(* IEC 61131-3 sources: POMIRTS_lab3/AS/Library_2/LoopCont/V2.12.0, 3 files *)

(* ---- LoopCont.typ ---- *)
(********************************************************************
 * COPYRIGHT (C) BERNECKER + RAINER, AUSTRIA, A-5142 EGGELSBERG
 ********************************************************************
 * Library: LoopCont
 * File: LoopCont.typ
 * Created: 11.11.2003
 ********************************************************************
 * Global data types of library LoopCont
 ********************************************************************)
TYPE
	lcCurveByPoints_TabEntry_type : STRUCT
		x	: INT ;
		y	: INT ;
	END_STRUCT;
	lcpid_addPar_typ : STRUCT
		y_autotune_on	: INT ;
		y_autotune_off	: INT ;
		t_autotune_max	: UDINT ;
		diff_dx_max	: INT ;
		diff_dt_max	: UDINT ;
		osc_nrPeriods	: UINT ;
		osc_minAmplitude	: INT ;
		optSwitches	: UINT ;
		dY_max	: REAL ;
		Tf_Tv	: REAL ;
		Kw	: REAL ;
		Kfbk	: REAL ;
		fbk_mode	: USINT ;
		d_mode	: USINT ;
		calc_mode	: USINT ;
	END_STRUCT;
	lcpid_internal_typ : STRUCT
		size	: UINT ;
		valid	: BOOL ;
		autotune_addpar	: lcpid_addPar_typ ;
		Y_max	: INT ;
		Y_min	: INT ;
		dY_max1	: DINT ;
		Kp1	: DINT ;
		Kp_Tn_1	: DINT ;
		Tv_Tf_1	: DINT ;
		Tf_reciproc_1	: DINT ;
		Kw1	: DINT ;
		Kfbk_Kp_1	: DINT ;
		fbk_mode	: USINT ;
		d_mode	: USINT ;
		calc_mode	: USINT ;
		prescalerPow2	: UINT ;
		force_outmode	: USINT ;
		Y_force	: INT ;
		W	: INT ;
		X	: INT ;
		pid_init	: USINT ;
		dt	: UDINT ;
		Yp1	: DINT ;
		Yp2	: DINT ;
		dYi1	: DINT ;
		dYi2	: DINT ;
		Yi1	: DINT ;
		Yi2	: DINT ;
		dt_Tf_1	: DINT ;
		a11	: DINT ;
		a12	: DINT ;
		a21	: DINT ;
		a22	: DINT ;
		Yd1	: DINT ;
		Yd2	: DINT ;
		Ytotal1	: DINT ;
		Ytotal2	: DINT ;
		Ylim1	: DINT ;
		Ylim2	: DINT ;
		Y1	: DINT ;
		Y2	: DINT ;
		e_fbk	: DINT ;
	END_STRUCT;
	lcpid_osc_val_typ : STRUCT
		X	: INT ;
		t	: UDINT ;
	END_STRUCT;
	lcpid_osc_per_typ : STRUCT
		max	: lcpid_osc_val_typ ;
		min	: lcpid_osc_val_typ ;
	END_STRUCT;
	lcpid_osc_typ : STRUCT
		i_maxPeriod	: UINT ;
		i_period	: UINT ;
		X_amplitude	: DINT ;
		amplitudeRatio	: REAL ;
		tPeriod	: UDINT ;
		period	: ARRAY[0..4] OF lcpid_osc_per_typ ;
	END_STRUCT;
	lcpid_procPar_typ : STRUCT
		size	: UINT ;
		stepResp_valid	: BOOL ;
		stepResp_v	: REAL ;
		stepResp_t_u	: UDINT ;
		osc_valid	: BOOL ;
		osc_amplitudeRatio	: REAL ;
		osc_tPeriod	: UDINT ;
		force_params	: BOOL ;
		Kp	: REAL ;
		Tn	: REAL ;
		Tv	: REAL ;
	END_STRUCT;
	lcpid_old_typ : STRUCT
		processPar	: lcpid_procPar_typ ;
		P_manualAdjust	: INT ;
		I_manualAdjust	: INT ;
		D_manualAdjust	: INT ;
		Y_min	: INT ;
		Y_max	: INT ;
		dY_max	: REAL ;
		Kw	: REAL ;
		Kfbk	: REAL ;
		enable	: BOOL ;
		request	: USINT ;
		time	: UDINT ;
	END_STRUCT;
	lcpid_stepResp_typ : STRUCT
		W_old	: INT ;
		dW	: INT ;
		x_prev	: INT ;
		x_inflectionPt	: INT ;
		t_inflectionPt	: UDINT ;
		v	: REAL ;
		v_max	: REAL ;
		t_u	: UDINT ;
		x_pre	: INT ;
		x_max	: INT ;
	END_STRUCT;
	lcpid_diff_typ : STRUCT
		init	: BOOL ;
		x_old	: INT ;
		dx	: INT ;
		dt	: UDINT ;
		dx_dt	: REAL ;
	END_STRUCT;
END_TYPE

(* ---- LoopCont.fun ---- *)
(********************************************************************
 * COPYRIGHT (C) BERNECKER + RAINER, AUSTRIA, A-5142 EGGELSBERG
 ********************************************************************
 * Library: LoopCont
 * File: LoopCont.fun
 * Created: 11.11.2003
 ********************************************************************
 * Functions and function blocks of library LoopCont
 ********************************************************************)
FUNCTION_BLOCK LCCurveByPoints
	VAR_INPUT
		x	:INT;
		NoOfPoints	:UINT;
		ptr_table	:REFERENCE TO lcCurveByPoints_TabEntry_type;
	END_VAR
	VAR_OUTPUT
		status	:UINT;
		y	:INT;
	END_VAR
	VAR
		i_tab	:INT;
		iterations	:UINT;
		scal1	:LCScINT;
	END_VAR
END_FUNCTION_BLOCK
FUNCTION_BLOCK LCPWM_DMod
	VAR_INPUT
		enable	:BOOL;
		x	:INT;
		max_value	:INT;
		min_value	:INT;
		tminpuls	:UINT;
		tperiod	:UINT;
		basetime	:UDINT;
	END_VAR
	VAR_OUTPUT
		status	:UINT;
		y	:BOOL;
	END_VAR
	VAR
		area	:DINT;
		period	:UINT;
		time_old	:UDINT;
		last	:UINT;
		x_old	:INT;
		enable_old	:BOOL;
	END_VAR
END_FUNCTION_BLOCK
FUNCTION_BLOCK LCPIDpara
	VAR_INPUT
		enable	:BOOL;
		enter	:BOOL;
		Y_max	:INT;
		Y_min	:INT;
		dY_max	:REAL;
		Kp	:REAL;
		Tn	:REAL;
		Tv	:REAL;
		Tf	:REAL;
		Kw	:REAL;
		Kfbk	:REAL;
		fbk_mode	:USINT;
		d_mode	:USINT;
		calc_mode	:USINT;
	END_VAR
	VAR_OUTPUT
		status	:UINT;
		ident	:UDINT;
	END_VAR
	VAR
		internal_data	:lcpid_internal_typ;
	END_VAR
END_FUNCTION_BLOCK
FUNCTION_BLOCK LCRampLim
	VAR_INPUT
		enable	:BOOL;
		x	:INT;
		tup	:UINT;
		tdown	:UINT;
		max_value	:INT;
		min_value	:INT;
		yset	:INT;
		set	:BOOL;
		basetime	:UDINT;
	END_VAR
	VAR_OUTPUT
		status	:UINT;
		y	:INT;
		xreached	:BOOL;
		max_limit	:BOOL;
		min_limit	:BOOL;
	END_VAR
	VAR
		time_old	:UDINT;
		rest	:UINT;
		enable_old	:BOOL;
	END_VAR
END_FUNCTION_BLOCK
FUNCTION_BLOCK LCPID
	VAR_INPUT
		enable	:BOOL;
		ident	:UDINT;
		W	:INT;
		X	:INT;
		A	:INT;
		Y_man	:INT;
		Y_fbk	:INT;
		hold_I	:BOOL;
		out_mode	:USINT;
		basetime	:UDINT;
	END_VAR
	VAR_OUTPUT
		status	:UINT;
		e	:DINT;
		Y	:INT;
		Yp	:DINT;
		Yi	:DINT;
		Yd	:DINT;
	END_VAR
	VAR
		time_old	:UDINT;
		Tv_Tf_old	:DINT;
		enable_old	:BOOL;
		e_old	:DINT;
	END_VAR
END_FUNCTION_BLOCK
FUNCTION_BLOCK LCTimeBasedOnOff
	VAR_INPUT
		enable	:BOOL;
		x	:INT;
		max_value	:INT;
		min_value	:INT;
		timpulse	:UINT;
		tchange_up	:UINT;
		tchange_dwn	:UINT;
		ref	:BOOL;
		basetime	:UDINT;
	END_VAR
	VAR_OUTPUT
		status	:UINT;
		up	:BOOL;
		down	:BOOL;
		hysteresis_up	:UINT;
		hysteresis_dwn	:UINT;
		refOK	:BOOL;
	END_VAR
	VAR
		time_old	:UDINT;
		ref_old	:BOOL;
		t_cnt	:DINT;
		y_fix31_1	:DINT;
		y_fix31_2	:DINT;
	END_VAR
END_FUNCTION_BLOCK
FUNCTION_BLOCK LCDifferentiate
	VAR_INPUT
		enable	:BOOL;
		x	:INT;
		tv	:UINT;
		tf	:UINT;
		basetime	:UDINT;
	END_VAR
	VAR_OUTPUT
		status	:UINT;
		y	:INT;
	END_VAR
	VAR
		time_old	:UDINT;
		enable_old	:BOOL;
		a2n	:DINT;
		a1	:DINT;
	END_VAR
END_FUNCTION_BLOCK
FUNCTION_BLOCK LCPIDAutoTune
	VAR_INPUT
		enable	:BOOL;
		Y_max	:INT;
		Y_min	:INT;
		P_manualAdjust	:INT;
		I_manualAdjust	:INT;
		D_manualAdjust	:INT;
		request	:USINT;
		basetime	:UDINT;
	END_VAR
	VAR_OUTPUT
		status	:UINT;
		ident	:UDINT;
		addInfo	:UINT;
		state	:UINT;
	END_VAR
	VAR
		dt	:UDINT;
		t_autotune	:UDINT;
		diff	:lcpid_diff_typ;
		old	:lcpid_old_typ;
		stepResponse	:lcpid_stepResp_typ;
		oscillation	:lcpid_osc_typ;
		processPar	:lcpid_procPar_typ;
		internal_data	:lcpid_internal_typ;
	END_VAR
END_FUNCTION_BLOCK
FUNCTION_BLOCK LC2PHy
	VAR_INPUT
		enable	:BOOL;
		x	:INT;
		xstart	:INT;
		xsetvalue	:INT;
		hysteresis	:UINT;
		ymax	:INT;
		ymin	:INT;
	END_VAR
	VAR_OUTPUT
		status	:UINT;
		y	:INT;
	END_VAR
	VAR
		y1	:BOOL;
		enable_old	:BOOL;
		x_old	:INT;
	END_VAR
END_FUNCTION_BLOCK
FUNCTION_BLOCK LCScUINT
	VAR_INPUT
		x	:UINT;
		x1	:UINT;
		y1	:UINT;
		x2	:UINT;
		y2	:UINT;
	END_VAR
	VAR_OUTPUT
		y	:UINT;
	END_VAR
END_FUNCTION_BLOCK
FUNCTION_BLOCK LC3PHy
	VAR_INPUT
		enable	:BOOL;
		x	:INT;
		xstart	:INT;
		xsetvalue1	:INT;
		xsetvalue2	:INT;
		hysteresis1	:UINT;
		hysteresis2	:UINT;
		ymax	:INT;
		ymid	:INT;
		ymin	:INT;
	END_VAR
	VAR_OUTPUT
		status	:UINT;
		y	:INT;
		ymx	:BOOL;
		ymn	:BOOL;
	END_VAR
	VAR
		enable_old	:BOOL;
		x_old	:INT;
	END_VAR
END_FUNCTION_BLOCK
FUNCTION_BLOCK LCComparator
	VAR_INPUT
		enable	:BOOL;
		xp	:INT;
		xn	:INT;
		sd	:UINT;
	END_VAR
	VAR_OUTPUT
		greater	:BOOL;
		equal	:BOOL;
		lower	:BOOL;
	END_VAR
END_FUNCTION_BLOCK
FUNCTION_BLOCK LCCounter
	VAR_OUTPUT
		muscnt	:UDINT;
		mus100cnt	:UDINT;
		mscnt	:UDINT;
		ms100cnt	:UDINT;
		seccnt	:UDINT;
	END_VAR
	VAR
		state	:UINT;
		sysinf_inst	:SysInfo;
		musecs_old	:UINT;
		bootkey_old	:UDINT;
		sys_ticks_old	:UDINT;
		to_100us	:UDINT;
		to_1ms	:UDINT;
		to_100ms	:UINT;
		to_1s	:UINT;
	END_VAR
END_FUNCTION_BLOCK
FUNCTION_BLOCK LCIntegrate
	VAR_INPUT
		enable	:BOOL;
		x	:INT;
		tn	:UINT;
		max_value	:INT;
		min_value	:INT;
		yset	:INT;
		set	:BOOL;
		basetime	:UDINT;
	END_VAR
	VAR_OUTPUT
		status	:UINT;
		y	:INT;
		max_limit	:BOOL;
		min_limit	:BOOL;
	END_VAR
	VAR
		time_old	:UDINT;
		rest	:DINT;
		enable_old	:BOOL;
	END_VAR
END_FUNCTION_BLOCK
FUNCTION_BLOCK LCLimit
	VAR_INPUT
		enable	:BOOL;
		in	:DINT;
		max_value	:INT;
		min_value	:INT;
	END_VAR
	VAR_OUTPUT
		status	:UINT;
		out	:INT;
		max_limit	:BOOL;
		min_limit	:BOOL;
	END_VAR
END_FUNCTION_BLOCK
FUNCTION_BLOCK LCLiScDINT
	VAR_INPUT
		x	:DINT;
		x1	:DINT;
		y1	:DINT;
		x2	:DINT;
		y2	:DINT;
	END_VAR
	VAR_OUTPUT
		y	:DINT;
	END_VAR
END_FUNCTION_BLOCK
FUNCTION_BLOCK LCLiScINT
	VAR_INPUT
		x	:INT;
		x1	:INT;
		y1	:INT;
		x2	:INT;
		y2	:INT;
	END_VAR
	VAR_OUTPUT
		y	:INT;
	END_VAR
END_FUNCTION_BLOCK
FUNCTION_BLOCK LCLiScUINT
	VAR_INPUT
		x	:UINT;
		x1	:UINT;
		y1	:UINT;
		x2	:UINT;
		y2	:UINT;
	END_VAR
	VAR_OUTPUT
		y	:UINT;
	END_VAR
END_FUNCTION_BLOCK
FUNCTION_BLOCK LCMovAvFilter
	VAR_INPUT
		enable	:BOOL;
		x	:INT;
		base	:UINT;
	END_VAR
	VAR_OUTPUT
		status	:UINT;
		y	:INT;
	END_VAR
	VAR
		sum_old	:DINT;
		x_old_ptr	:UDINT;
		x_old	:ARRAY[0..31] OF INT;
		xIdx	:UINT;
		base_old	:UINT;
		enable_old	:BOOL;
		bootkey_old	:UDINT;
	END_VAR
END_FUNCTION_BLOCK
FUNCTION_BLOCK LCNegDINT
	VAR_INPUT
		in	:DINT;
	END_VAR
	VAR_OUTPUT
		out	:DINT;
	END_VAR
END_FUNCTION_BLOCK
FUNCTION_BLOCK LCNegINT
	VAR_INPUT
		in	:INT;
	END_VAR
	VAR_OUTPUT
		out	:INT;
	END_VAR
END_FUNCTION_BLOCK
FUNCTION_BLOCK LCNegPeakVal
	VAR_INPUT
		in	:INT;
		reset	:BOOL;
	END_VAR
	VAR_OUTPUT
		out	:INT;
	END_VAR
END_FUNCTION_BLOCK
FUNCTION_BLOCK LCPosPeakVal
	VAR_INPUT
		in	:INT;
		reset	:BOOL;
	END_VAR
	VAR_OUTPUT
		out	:INT;
	END_VAR
END_FUNCTION_BLOCK
FUNCTION_BLOCK LCPT1
	VAR_INPUT
		enable	:BOOL;
		x	:INT;
		t	:UINT;
		yset	:INT;
		set	:BOOL;
		basetime	:UDINT;
	END_VAR
	VAR_OUTPUT
		status	:UINT;
		y	:INT;
	END_VAR
	VAR
		time_old	:UDINT;
		rest	:DINT;
		enable_old	:BOOL;
	END_VAR
END_FUNCTION_BLOCK
FUNCTION_BLOCK LCScDINT
	VAR_INPUT
		x	:DINT;
		x1	:DINT;
		y1	:DINT;
		x2	:DINT;
		y2	:DINT;
	END_VAR
	VAR_OUTPUT
		y	:DINT;
	END_VAR
END_FUNCTION_BLOCK
FUNCTION_BLOCK LCScINT
	VAR_INPUT
		x	:INT;
		x1	:INT;
		y1	:INT;
		x2	:INT;
		y2	:INT;
	END_VAR
	VAR_OUTPUT
		y	:INT;
	END_VAR
END_FUNCTION_BLOCK

(* ---- LoopCont.var ---- *)
(********************************************************************
 * COPYRIGHT (C) BERNECKER + RAINER, AUSTRIA, A-5142 EGGELSBERG
 ********************************************************************
 * Library: LoopCont
 * File: LoopCont.var
 * Created: 11.11.2003
 ********************************************************************
 * Constants of library LoopCont
 ********************************************************************)
VAR CONSTANT
	LCPIDAUTOTUNE_STATE_STEPRESPONSE	: UINT	:= 20;
	LCPIDAUTOTUNE_ADDINFO_OSC_PERIOD	: UINT	:= 101;
	LCPIDAUTOTUNE_STATE_RESET_CTRLR	: UINT	:= 49;
	LCPIDAUTOTUNE_REQU_STEPRESPONSE	: USINT	:= 1;
	LCPIDAUTOTUNE_ADDINFO_PRESCALER	: UINT	:= 102;
	LC_ERR_LCPIDAutotune_W_CHANGED	: UINT	:= 12041;
	LC_ERR_LCPIDAutotune_PARAMETER	: UINT	:= 12039;
	LCPID_OUT_MODE_FREEZE_JOLTFREE	: UINT	:= 105;
	LCPIDAUTOTUNE_ADDINFO_OSC_AMPL	: UINT	:= 100;
	LC_ERR_LCTimBasOnOff_TIMPULSE	: UINT	:= 12036;
	LCPID_OUT_MODE_CLOSE_JOLTFREE	: UINT	:= 104;
	LCPIDAUTOTUNE_STATE_WAIT_STEP	: UINT	:= 10;
	LCPIDAUTOTUNE_STATE_OSCILLATE	: UINT	:= 40;
	LC_ERR_LCTimBasOnOff_TCHANGE	: UINT	:= 12035;
	LC_ERR_LCPIDAutotune_TIMEOUT	: UINT	:= 12040;
	LC_ERR_LCCurveByPoints_TABLE	: UINT	:= 12045;
	LCPID_OUT_MODE_OPEN_JOLTFREE	: UINT	:= 103;
	LCPIDAUTOTUNE_STATE_WAIT_MAX	: UINT	:= 30;
	LCPIDAUTOTUNE_STATE_FINISHED	: UINT	:= 50;
	LCPIDAUTOTUNE_REQU_OSCILLATE	: USINT	:= 2;
	LCPID_OUT_MODE_MAN_JOLTFREE	: USINT	:= 102;
	LCPID_FBK_MODE_EXT_SELECTOR	: USINT	:= 3;
	LCPIDAUTOTUNE_REQU_AUTOTUNE	: USINT	:= 3;
	LCPIDAUTOTUNE_ADDINFO_Y_OFF	: UINT	:= 103;
	LC_ERR_LCRampLim_TUP_TDOWN	: UINT	:= 12034;
	LC_ERR_LCPWM_DMod_TMINPULS	: UINT	:= 12032;
	LC_ERR_LCPID_PAR_PRESCALER	: UINT	:= 12042;
	LC_ERR_LCPIDAutotune_ABORT	: UINT	:= 12038;
	LCPIDAUTOTUNE_ADDINFO_Y_ON	: UINT	:= 104;
	LC_ERR_LCPWM_DMod_TPERIOD	: UINT	:= 12033;
	LC_ERR_LCPID_PAR_CALCMODE	: UINT	:= 12021;
	LC_ERR_LCMovAvFilter_BASE	: UINT	:= 12017;
	LCPIDAUTOTUNE_STATE_READY	: UINT	:= 0;
	LC_WARN_LCPID_YFBK_LIMIT	: UINT	:= 12003;
	LC_WARN_LCPID_I_MINLIMIT	: UINT	:= 12002;
	LC_WARN_LCPID_I_MAXLIMIT	: UINT	:= 12001;
	LC_ERR_LCPID_PAR_FBKMODE	: UINT	:= 12024;
	LC_ERR_LC3PHy_XSETVALUE	: UINT	:= 12015;
	LC_ERR_LCPID_PAR_DYMAX	: UINT	:= 12023;
	LC_ERR_LCPID_PAR_DMODE	: UINT	:= 12022;
	LCPIDAUTOTUNE_REQU_OFF	: USINT	:= 0;
	LC_WARN_LCxPHy_XSTART	: UINT	:= 12006;
	LC_ERR_LCPID_PAR_KFBK	: UINT	:= 12025;
	LC_ERR_LCIntegrate_TN	: UINT	:= 12016;
	LCPID_OUT_MODE_FREEZE	: USINT	:= 5;
	LCPID_FBK_MODE_INTERN	: USINT	:= 1;
	LCPID_FBK_MODE_EXTERN	: USINT	:= 2;
	LCPID_CALC_MODE_EXACT	: USINT	:= 1;
	LC_ERR_LCPID_PARADAT	: UINT	:= 12020;
	LC_ERR_LCPID_OUTMODE	: UINT	:= 12019;
	LCPID_OUT_MODE_CLOSE	: USINT	:= 4;
	LCPID_CALC_MODE_FAST	: USINT	:= 2;
	LC_WARN_DT_MAXLIMIT	: UINT	:= 12000;
	LC_ERR_LCPID_PAR_TV	: UINT	:= 12030;
	LC_ERR_LCPID_PAR_TN	: UINT	:= 12029;
	LC_ERR_LCPID_PAR_TF	: UINT	:= 12028;
	LC_ERR_LCPID_PAR_KW	: UINT	:= 12027;
	LC_ERR_LCPID_PAR_KP	: UINT	:= 12026;
	LCPID_OUT_MODE_OPEN	: USINT	:= 3;
	LCPID_OUT_MODE_AUTO	: USINT	:= 1;
	LC_ERR_LCPID_IDENT	: UINT	:= 12018;
	LCPID_OUT_MODE_MAN	: USINT	:= 2;
	LC_ERR_DISABLED	: UINT	:= 65534;
	LC_ERR_LCPT1_T	: UINT	:= 12031;
	LCPID_D_MODE_X	: USINT	:= 1;
	LCPID_D_MODE_E	: USINT	:= 2;
	LC_WARN_Tx_DT	: UINT	:= 12007;
	LC_ERR_MAXMIN	: UINT	:= 12037;
	LC_ERROR	: UINT	:= 12015;
END_VAR
